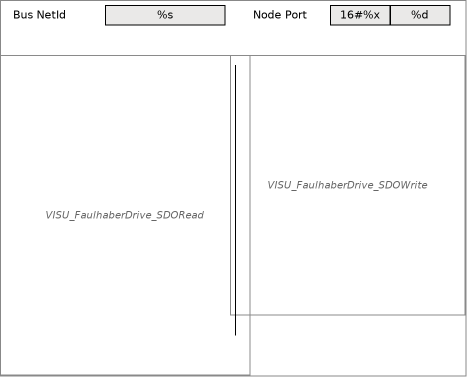
VISUALIZATION VISU_FaulhaberDrive  // 467x377
VAR_IN_OUT
	drive : FaulhaberDrive;
    widget : FaulhaberDriveWidget;
END_VAR
    Frame (0,55 250x320)
        shows VISU_FaulhaberDrive_SDORead(drive := drive, widget := widget)
    Label (10,0 80x30), "Bus NetId"
    Rectangle (105,5 120x20), "%s", text variable: drive.config.CANopenBusNetId
    Rectangle (330,5 60x20), "16#%x", text variable: drive.config.CANopenNodePort
    Label (250,0 80x30), "Node Port"
    Rectangle (390,5 60x20), "%d", text variable: drive.config.CANopenNodePort
    Frame (230,55 235x260)
        shows VISU_FaulhaberDrive_SDOWrite(drive := drive, widget := widget)
    Line (235,65) (235,335)
END_VISUALIZATION

(* stored: Version 1.1.0.1, ProductVersion 3.1.4019.2
   Visu VISU_FaulhaberDrive: Id {42edd0b3-ecba-4027-975c-6e8ab394416d} *)
